// TIA Portal V21 export
TYPE "TipoDatiVuoto"
   STRUCT
      EmptyBool : Bool;
   END_STRUCT;
END_TYPE
